(* PLC project static_torsion.project, CODESYS CODESYS V3.5 SP17 Patch 3 *)
(* stored: creationDateTime 1970-01-01T00:00:00, modificationDateTime 2026-06-22T15:12:39.4699931 *)

FUNCTION CalculateScaledTorque : INT
  VAR_INPUT
    torque : REAL;
  END_VAR
  VAR CONSTANT
    scale_ : REAL := 500;
  END_VAR

            CalculateScaledTorque:= LIMIT(-32768, TO_INT(torque * scale_), 32767);
          
END_FUNCTION
